TYPE Pump EXTENDS Valve :
STRUCT
	nPulse : INT;
	sTime : STRING;
	sRemainingTime : STRING;
END_STRUCT
END_TYPE

(* stored: Version 1.1.0.1, ProductVersion 3.1.4024.3
   DUT Pump: Id {08f99879-e236-4ab2-8842-35ebc829f669} *)
